KUKA KRL data list: AprilTag.dat

&ACCESS RVP
&PARAM EDITMASK = *
DEFDAT AprilTag

   ;FOLD EXTERNAL DECLARATIONS;%{PE}%MKUKATPBASIS,%CEXT,%VCOMMON,%P
   ;FOLD BASISTECH EXT;%{PE}%MKUKATPBASIS,%CEXT,%VEXT,%P
   EXT  BAS (BAS_COMMAND  :IN,REAL  :IN )
   ;ENDFOLD (BASISTECH EXT)
   ;FOLD USER EXT;%{E}%MKUKATPUSER,%CEXT,%VEXT,%P
   ;Make your modifications here

   ; Common structures and variables
   STRUC RETURNCODE_T INT VALUE,CHAR MSG[512]
   DECL INT RCEkiAliveFlagNo=997
   DECL RETURNCODE_T RETURNCODE
   DECL FRAME POSE_IDENT={X 0.0,Y 0.0,Z 0.0,A 0.0,B 0.0,C 0.0}

   ; Service configuration
   DECL CHAR serviceNameDetect[64]

   ; Detection results
   DECL FRAME DETECTEDTAGS[32]
   DECL INT NUMDETECTEDTAGS

   ; Frame data
   DECL FDAT FP1={TOOL_NO 4,BASE_NO 0,IPO_FRAME #BASE,POINT2[] " "}

   ; Point data
   DECL PDAT PPDAT1={VEL 100.0,ACC 100.0,APO_DIST 100.0,APO_MODE #CPTP,GEAR_JERK 50.0,EXAX_IGN 0}

   ; Start position
   DECL E6POS STARTPOSE={X 0,Y 0,Z 0,A 0,B 0,C 0,S 0,T 0,E1 0.0,E2 0.0,E3 0.0,E4 0.0,E5 0.0,E6 0.0}

   ; Movement data
   DECL LDAT lDatDefault={VEL 2.00000,ACC 20.0000,APO_DIST 10.0000,APO_FAC 50.0000,AXIS_VEL 100.000,AXIS_ACC 100.000,ORI_TYP #VAR,CIRC_TYP #BASE,JERK_FAC 50.0000,GEAR_JERK 100.000,EXAX_IGN 0,CB {AUX_PT {ORI #CONSIDER,E1 #CONSIDER,E2 #CONSIDER,E3 #CONSIDER,E4 #CONSIDER,E5 #CONSIDER,E6 #CONSIDER},TARGET_PT {ORI #INTERPOLATE,E1 #INTERPOLATE,E2 #INTERPOLATE,E3 #INTERPOLATE,E4 #INTERPOLATE,E5 #INTERPOLATE,E6 #INTERPOLATE}}}
   DECL FDAT fDatDefault={TOOL_NO 4,BASE_NO 0,IPO_FRAME #BASE,POINT2[] " "}
   DECL PDAT pDatDefault={VEL 10.0000,ACC 20.0000,APO_DIST 10.0000,APO_MODE #CDIS,GEAR_JERK 100.000,EXAX_IGN 0}

   ;ENDFOLD (USER EXT)
   ;ENDFOLD (EXTERNAL DECLARATIONS)
ENDDAT
